PROGRAM INTERNAL PRG_TESTS

(* Instantiate test suites here. Naming convention for tests should be a suffix with _Tests.
Good practice for creating test methods is to end them with _test as well. *)

VAR
	EndurancePyrometer_Tests			: FB_EndurancePyrometer_Tests;
	EndurancePyrometerConstants_Tests	: FB_EndurancePyrometerConstants_Tests;
END_VAR

// Run tests in parallel
//TcUnit.RUN();

// Run tests in sequence, one after the other.
TcUnit.RUN_IN_SEQUENCE();

END_PROGRAM

(* stored: Version 1.1.0.1, ProductVersion 3.1.4024.16
   POU PRG_TESTS: Id {dd239b23-fd06-45c2-8d55-97bc3cfa2578}, SpecialFunc None *)
